FUNCTION_BLOCK Festo_IoLink_VacumEjector_OVEM_H_CE
VAR_INPUT
     ReadParameters  : BOOL;             // Read parameters - starts on rising trigger 
     WriteParameters : BOOL;             // Set parameters  - starts on rising trigger
     Reset           : BOOL;             // Reset application  - Reset sequence. 
     ApplicationTag  : STRING(32) := ''; // Application Tag to be writen to IO Link Device 
     AirSaveFunction : BOOL;             // Parameter Air Safe function
     AutoDropTime    : UINT;             // Auto drop time - 0x0198 - default Value: 80
     AmsNetID        : AMSNETID;         // AoeNetId from IO link terminal    
     Port            : UINT;             // Port on IO link terminal 
     Name            : STRING(255);      // Name of IO link device ??
END_VAR
VAR_OUTPUT
     Busy                : BOOL := FALSE;
     Done                : BOOL := FALSE;
     Error               : BOOL := FALSE;
     ProductId           : STRING;
     ApplicationTagRead  : STRING(32) := '';
     AirSaveFunctionRead : BOOL; // Air safe function 
     ParametersRead      : BOOL; // if this i ok, the parameters is read

     AutoDropTimeRead : INT; // 0x0198 - 80 
     AdsError         : E_AdsErr    := E_AdsErr.NOERR;
     IolError         : E_IolError  := E_IolError.NoError;
     ErrorTxt         : STRING(255) := '';
END_VAR
VAR
     _InitDone           : BOOL := FALSE;
     _ReadParameters     : BOOL; // Read parameters
     _SetParameters      : BOOL; // Set parameters
     _ApplicationTagRead : STRING(32) := '';
     _fbIolSlave         : FB_IolStdVarSlave;
     _fbIolVarSlave      : FB_IolSlave;
     _hr                 : HRESULT;
     _State              : INT; // case state	
     _rtReadParameter    : R_TRIG;
     _rtWriteParameter   : R_TRIG;

END_VAR


// Triggers for start sequence.
_rtReadParameter(CLK := ReadParameters);
_rtWriteParameter(CLK := WriteParameters);

CASE _State OF

     00: //Init 
          _fbIolSlave.MasterAoeNetId := F_CreateAmsNetId(AmsNetID); //Creates NETID String
          _fbIolSlave.Port           := Port;
          _fbIolSlave.Name           := Name;
          _State                     := 10;


     10: // Idle

          IF _rtReadParameter.Q THEN
               _State := 20;
          ELSIF _rtWriteParameter.Q THEN
               _State := 120;
          END_IF

     20: // Read Parameters 
          // Read Application Tag

          _hr := _fbIolSlave.ReadApplicationSpecificTag(ApplicationTagRead);

          IF NOT F_IolIsBusy(_hr) THEN
               IF FAILED(_hr) THEN
                    Busy       := FALSE;
                    Error      := TRUE;
                    ErrorTxt   := _fbIolSlave.ErrorTxt; // TODO
                    AdsError   := F_IolGetAdsError(_hr);
                    IolError   := F_IolGetIolError(_hr);
                    _State := 999; // Error;
               ELSE
                    _State := 30; // CHECK;
               END_IF
          END_IF
		30: // Read



     999: // Error state 

          IF Reset THEN
               Busy     := FALSE;
               Error    := FALSE;
               AdsError := E_AdsErr.NOERR;
               IolError := E_IolError.NoError;
               ErrorTxt := '';
          END_IF
END_CASE

METHOD PRIVATE ReadApplicationTag : UDINT
VAR_INPUT 
	Execute : BOOL; 
END_VAR
////
// FB State Machine
//
CASE _ReadState OF

     // IDLE
     0: ;

          IF Execute THEN
               _ReadState := 10;
          END_IF

     10: // Read application Tag

          _hr := _fbIolSlave.ReadApplicationSpecificTag(ApplicationTagRead);

          IF NOT F_IolIsBusy(_hr) THEN
               IF FAILED(_hr) THEN
                    Busy       := FALSE;
                    Error      := TRUE;
                    ErrorTxt   := _fbIolSlave.ErrorTxt; // TODO
                    AdsError   := F_IolGetAdsError(_hr);
                    IolError   := F_IolGetIolError(_hr);
                    _ReadState := 999; // Error;
               ELSE
                    _ReadState := 30; // CHECK;
               END_IF
          END_IF

     // CHECK
     30: IF ApplicationTag <> _ApplicationTagRead THEN
               Busy     := FALSE;
               Error    := TRUE;
               ErrorTxt := 'sApplicationTag and sApplicationTagRead are not equal!';
          ELSE
               Busy := FALSE;
               Done := TRUE;
               //              _ReadState := 0;
          END_IF

     999: // Error state

          IF NOT Execute THEN

               _hr := _fbIolSlave.SysCmdApplicationReset();

               IF NOT F_IolIsBusy(_hr) THEN
                    IF FAILED(_hr) THEN
                         Busy     := FALSE;
                         Error    := TRUE;
                         ErrorTxt := _fbIolSlave.ErrorTxt; 
                         AdsError := F_IolGetAdsError(_hr);
                         IolError := F_IolGetIolError(_hr);
                         //_ReadState := 999; // Error;
                    ELSE
                         _ReadState := 0; // CHECK;
                    END_IF
               END_IF

          END_IF

END_CASE

////
// call FBs
//
_fbIolSlave();
END_METHOD

METHOD PRIVATE WriteApplicationTag : UDINT
VAR_INPUT
END_VAR
END_METHOD

END_FUNCTION_BLOCK

(* stored: Version 1.1.0.1, ProductVersion 3.1.4024.11
   POU Festo_IoLink_VacumEjector_OVEM_H_CE: Id {b6245ee7-b1b9-443b-84b3-5d7151a3bb6b}, SpecialFunc None
   Method ReadApplicationTag: Id {b0d51dd5-7959-4151-a6db-a6937abebc2d}
   Method WriteApplicationTag: Id {0004d753-af26-41e9-a2f2-32c49d39e4f1} *)
